// TIA Portal V18 export
// export: Created 2026-03-12T15:56:19.3011542Z, ExportSetting WithDefaults, DisplayName Totally Integrated Automation Portal, DisplayVersion V18 Update 5, DisplayName TIA Portal Openness, DisplayVersion V18 Update 5, DisplayName TIA Portal Version Control Interface, DisplayVersion V18, DisplayName SINAMICS Startdrive Advanced, DisplayVersion V18, DisplayName SINAMICS Startdrive G130, G150, S120, S150, SINAMICS MV, S210, DisplayVersion V18, DisplayName SINAMICS Startdrive G110M, G120, G120C, G120D, G120P, G115D, DisplayVersion V18, DisplayName STEP 7 Professional, DisplayVersion V18 Update 5, DisplayName STEP 7 Safety, DisplayVersion V18, DisplayName WinCC Professional, DisplayVersion V18 Update 5
DATA_BLOCK "FB_HORÍMETRO BH-01A"   // DB215
VERSION : 0.1
// stored: AutoNumber true, DBAccessibleFromOPCUA true, DBAccessibleFromWebserver true, InstanceOfName FB_HORÍMETRO, InstanceOfType FB
"FB_HORÍMETRO"
   // VAR_INPUT
   //    INPUT_LIGADO : Bool;
   //    INPUT_RESET_HORIMETRO : Bool;
   // END_VAR
   // VAR_IN_OUT
   //    HORIMETRO : UInt;
   // END_VAR
   // VAR RETAIN
   //    RESET_SEGUNDO : Bool;
   //    MINUTO : Bool;
   //    COUNT_MINUTO : Bool;
   //    RESET_MINUTO : Bool;
   //    HORA : Bool;
   //    COUNT_HORA : Bool;
   //    HORAS : UInt;
   //    TIMER_SEGUNDO : IEC_COUNTER;
   //    TIMER_MINUTO : IEC_COUNTER;
   // END_VAR
BEGIN
END_DATA_BLOCK
